// TIA Portal V19 export
TYPE "LEXCHANGETRAY_typeNgStrapConfigeration"
TITLE = exchangeTray_typeNgStrapConfigeration
// exchangeTray_typeNgStrapConfigeration related values
// stored: Access Published
   STRUCT
      referenceDesignator { S7_SetPoint := 'True'} : String[20] := 'NgStrap.';   // Device name or device ID
      simActive { S7_SetPoint := 'True'} : Bool := False;   // Simulation active
      refCount { S7_SetPoint := 'True'} : Int := 5;   // Reference count
   END_STRUCT;
END_TYPE
